FUNCTION_BLOCK FB_AlarmHandler EXTENDS FB_TcAlarm

VAR_INPUT
	evtEntry	: TcEventEntry;
	bEvt		: BOOL;
	bConfirm	: BOOL;
	sSystem		: STRING; // Adding Alarm system name
	sMessage	: STRING; // Alarm Message
END_VAR

VAR_OUTPUT
	
END_VAR

VAR
	bInit	: BOOL := TRUE;
	bMem	: BOOL;
	
END_VAR

IF bInit THEN
	SUPER^.CreateEx(evtEntry, TRUE, 0);
	bInit	:= FALSE;
END_IF

// To when the alarm is triggered for the first time
IF bEvt AND NOT bMem AND SUPER^.eConfirmationState <> TcEventConfirmationState.WaitForConfirmation THEN
	SUPER^.ipArguments.AddString(sSystem).AddString(sMessage); // Adiciona as strings ao alarme
	SUPER^.Raise(0);
END_IF

// To when the alarm is reset
IF bMem AND NOT bEvt THEN
	SUPER^.Clear(0, FALSE);
END_IF

// Alarm confirmation
IF bConfirm THEN
	SUPER^.Confirm(0);
END_IF

bMem := bEvt;

END_FUNCTION_BLOCK

(* stored: Version 1.1.0.1, ProductVersion 3.1.4024.12
   POU FB_AlarmHandler: Id {5e7f237a-32b2-4825-a094-3cb12ffb08a5}, SpecialFunc None *)
